FUNCTION_BLOCK ABSTRACT FastAttenuationBase EXTENDS TExecution IMPLEMENTS IDevice
VAR_INPUT
END_VAR
VAR_OUTPUT
END_VAR
VAR
	{attribute 'OPC.UA.DA' := '0'}
	_name : STRING;
	{attribute 'OPC.UA.DA' := '0'}
	_deviceID : STRING;					
	{attribute 'OPC.UA.DA' := '0'}
	_family : DeviceFamily;				
	{attribute 'OPC.UA.DA' := '0'}
	_logger : Logger;
	{attribute 'OPC.UA.DA' := '0'}
	_message : StringBuilder;	
	{attribute 'OPC.UA.DA' := '0'}
	_fastAttenuationConfig : DeviceConfiguration;
END_VAR

PROPERTY DeviceID : STRING
GET
DeviceID := _deviceID;
END_GET
SET
_deviceID := DeviceID;
END_SET
END_PROPERTY

PROPERTY Family : DeviceFamily
GET
Family := _family;
END_GET
SET
_family := Family;
END_SET
END_PROPERTY

METHOD PROTECTED ABSTRACT MoveAbsPosition
VAR_INPUT
	Execute : BOOL;
	AnglePosition : LREAL;
END_VAR
END_METHOD

PROPERTY Name : STRING
GET
Name := _name;
END_GET
SET
_name := Name;
END_SET
END_PROPERTY

END_FUNCTION_BLOCK

(* stored: Version 1.1.0.1, ProductVersion 3.1.4024.4
   POU FastAttenuationBase: Id {967127ee-a1aa-4917-8492-cbd328448d2e}, SpecialFunc None
   Property DeviceID: Id {a438fe7f-f069-49a8-a2a1-1b10ede6c220}
   Get Get: Id {75c3ad93-543c-44b9-8fa2-a7ee892dce9d}
   Set Set: Id {b657e510-10b3-4628-8c43-4d76d49dfe9d}
   Property Family: Id {1348c67c-a1be-4090-9855-b842e8c60dbd}
   Get Get: Id {87e2a58c-c839-4273-868a-4e6f3f82ced7}
   Set Set: Id {58c855e4-ad5f-4fd6-84a2-48a4770b874d}
   Method MoveAbsPosition: Id {f01d21fa-d485-458e-88c8-bc2e328e8a37}
   Property Name: Id {8aea5495-b46f-4a5a-ad8f-76d1e0f91a5a}
   Get Get: Id {26124808-f74f-4799-bde9-87f75b37edc3}
   Set Set: Id {3efde58d-a5d4-4efa-aae1-9059474710f0} *)
